FUNCTION exARRAY_MAX : REAL
VAR_INPUT
	pt: POINTER TO ARRAY[0..32000] OF REAL;
	size: UINT;
END_VAR
VAR
	i: UINT;
	stop: UINT;
END_VAR

stop := (size -SIZEOF(pt)) / SIZEOF(pt);
exARRAY_MAX := pt^[0];
FOR i := 1 TO stop DO
	IF pt^[i] > exARRAY_MAX THEN exARRAY_MAX := pt^[i]; END_IF;
END_FOR;

(* revision history
hm	2. oct 2006		rev 1.0
	original version

hm	16. mar. 2008	rev 1.1
	changed input size to uint
*)

END_FUNCTION

(* stored: Version 1.1.0.1, ProductVersion 3.1.4024.3
   POU exARRAY_MAX: Id {830dde70-9910-410c-94e3-1e39be3f3690}, SpecialFunc None *)
